(* IEC 61131-3 sources: lpmlv2022/test, 9 files *)

(* ---- test.st ---- *)
USING AxUnit.Assert;

NAMESPACE Simatic.Ax.lpmlv2022.Tests
    {TestFixture}
    CLASS MyTestFixture
        {Test}
        METHOD PUBLIC MyTestMethod
            Equal(actual := TRUE, expected := TRUE);
        END_METHOD
    END_CLASS
END_NAMESPACE

(* ---- TestConfigureCompleteCmdCfg.st ---- *)
USING AxUnit;
USING Simatic.Ax.LPMLV2022;

NAMESPACE Simatic.Ax.LPMLV2022.Tests

    {TestFixture}
    CLASS TestConfigureCompleteCmdCfg

        {Test}
        METHOD PUBLIC TestOnlySuspended
            VAR_TEMP
                result : DWORD;
            END_VAR

            ConfigureCompleteCmdCfg(
                Suspended := TRUE,
                Execute := FALSE,
                Held := FALSE,
                completeCmdCfg => result);

            Assert.Equal(actual := result.%X5, expected := TRUE);
            Assert.Equal(actual := result.%X6, expected := FALSE);
            Assert.Equal(actual := result.%X11, expected := FALSE);
            // Verify expected DWORD value (bit 5 set = 2^5 = 32 = 16#20)
            Assert.Equal(actual := result, expected := DWORD#16#0000_0020);

        END_METHOD

        {Test}
        METHOD PUBLIC TestOnlyExecute
            VAR_TEMP
                result : DWORD;
            END_VAR

            ConfigureCompleteCmdCfg(
                Suspended := FALSE,
                Execute := TRUE,
                Held := FALSE,
                completeCmdCfg => result);

            Assert.Equal(actual := result.%X5, expected := FALSE);
            Assert.Equal(actual := result.%X6, expected := TRUE);
            Assert.Equal(actual := result.%X11, expected := FALSE);
            // Verify expected DWORD value (bit 6 set = 2^6 = 64 = 16#40)
            Assert.Equal(actual := result, expected := DWORD#16#0000_0040);

        END_METHOD

        {Test}
        METHOD PUBLIC TestOnlyHeld
            VAR_TEMP
                result : DWORD;
            END_VAR

            ConfigureCompleteCmdCfg(
                Suspended := FALSE,
                Execute := FALSE,
                Held := TRUE,
                completeCmdCfg => result);

            Assert.Equal(actual := result.%X5, expected := FALSE);
            Assert.Equal(actual := result.%X6, expected := FALSE);
            Assert.Equal(actual := result.%X11, expected := TRUE);
            // Verify expected DWORD value (bit 11 set = 2^11 = 2048 = 16#800)
            Assert.Equal(actual := result, expected := DWORD#16#0000_0800);

        END_METHOD

        {Test}
        METHOD PUBLIC TestSuspendedAndExecute
            VAR_TEMP
                result : DWORD;
            END_VAR

            ConfigureCompleteCmdCfg(
                Suspended := TRUE,
                Execute := TRUE,
                Held := FALSE,
                completeCmdCfg => result);

            Assert.Equal(actual := result.%X5, expected := TRUE);
            Assert.Equal(actual := result.%X6, expected := TRUE);
            Assert.Equal(actual := result.%X11, expected := FALSE);
            // Verify expected DWORD value (bits 5+6 set = 32+64 = 96 = 16#60)
            Assert.Equal(actual := result, expected := DWORD#16#0000_0060);

        END_METHOD

        {Test}
        METHOD PUBLIC TestSuspendedAndHeld
            VAR_TEMP
                result : DWORD;
            END_VAR

            ConfigureCompleteCmdCfg(
                Suspended := TRUE,
                Execute := FALSE,
                Held := TRUE,
                completeCmdCfg => result);

            Assert.Equal(actual := result.%X5, expected := TRUE);
            Assert.Equal(actual := result.%X6, expected := FALSE);
            Assert.Equal(actual := result.%X11, expected := TRUE);
            // Verify expected DWORD value (bits 5+11 set = 32+2048 = 2080 = 16#820)
            Assert.Equal(actual := result, expected := DWORD#16#0000_0820);

        END_METHOD

        {Test}
        METHOD PUBLIC TestExecuteAndHeld
            VAR_TEMP
                result : DWORD;
            END_VAR

            ConfigureCompleteCmdCfg(
                Suspended := FALSE,
                Execute := TRUE,
                Held := TRUE,
                completeCmdCfg => result);

            Assert.Equal(actual := result.%X5, expected := FALSE);
            Assert.Equal(actual := result.%X6, expected := TRUE);
            Assert.Equal(actual := result.%X11, expected := TRUE);
            // Verify expected DWORD value (bits 6+11 set = 64+2048 = 2112 = 16#840)
            Assert.Equal(actual := result, expected := DWORD#16#0000_0840);

        END_METHOD

        {Test}
        METHOD PUBLIC TestAllStatesEnabled
            VAR_TEMP
                result : DWORD;
            END_VAR

            ConfigureCompleteCmdCfg(
                Suspended := TRUE,
                Execute := TRUE,
                Held := TRUE,
                completeCmdCfg => result);

            Assert.Equal(actual := result.%X5, expected := TRUE);
            Assert.Equal(actual := result.%X6, expected := TRUE);
            Assert.Equal(actual := result.%X11, expected := TRUE);
            // Verify expected DWORD value (bits 5+6+11 set = 32+64+2048 = 2144 = 16#860)
            Assert.Equal(actual := result, expected := DWORD#16#0000_0860);

        END_METHOD

        {Test}
        METHOD PUBLIC TestAllStatesDisabled
            VAR_TEMP
                result : DWORD;
            END_VAR

            ConfigureCompleteCmdCfg(
                Suspended := FALSE,
                Execute := FALSE,
                Held := FALSE,
                completeCmdCfg => result);

            Assert.Equal(actual := result.%X5, expected := FALSE);
            Assert.Equal(actual := result.%X6, expected := FALSE);
            Assert.Equal(actual := result.%X11, expected := FALSE);
            // Verify expected DWORD value (no bits set = 0)
            Assert.Equal(actual := result, expected := DWORD#16#0000_0000);

        END_METHOD

        {Test}
        METHOD PUBLIC TestUnusedBitsRemainZero
            VAR_TEMP
                result : DWORD;
                i : INT;
            END_VAR

            ConfigureCompleteCmdCfg(
                Suspended := TRUE,
                Execute := TRUE,
                Held := TRUE,
                completeCmdCfg => result);

            // Test that only the expected bits (5, 6, 11) are set
            // and all other bits remain 0
            FOR i := 0 TO 31 DO
                IF i = 5 OR i = 6 OR i = 11 THEN
                    // These bits should be TRUE
                    CONTINUE;
                ELSE
                    // All other bits should be FALSE
                    CASE i OF
                        0: Assert.Equal(actual := result.%X0, expected := FALSE);
                        1: Assert.Equal(actual := result.%X1, expected := FALSE);
                        2: Assert.Equal(actual := result.%X2, expected := FALSE);
                        3: Assert.Equal(actual := result.%X3, expected := FALSE);
                        4: Assert.Equal(actual := result.%X4, expected := FALSE);
                        7: Assert.Equal(actual := result.%X7, expected := FALSE);
                        8: Assert.Equal(actual := result.%X8, expected := FALSE);
                        9: Assert.Equal(actual := result.%X9, expected := FALSE);
                        10: Assert.Equal(actual := result.%X10, expected := FALSE);
                        12: Assert.Equal(actual := result.%X12, expected := FALSE);
                        13: Assert.Equal(actual := result.%X13, expected := FALSE);
                        14: Assert.Equal(actual := result.%X14, expected := FALSE);
                        15: Assert.Equal(actual := result.%X15, expected := FALSE);
                        // Testing a few more significant bits
                        16: Assert.Equal(actual := result.%X16, expected := FALSE);
                        20: Assert.Equal(actual := result.%X20, expected := FALSE);
                        31: Assert.Equal(actual := result.%X31, expected := FALSE);
                    END_CASE;
                END_IF;
            END_FOR;

        END_METHOD
    END_CLASS

END_NAMESPACE

(* ---- TestConfigureDisabledStatesCfg.st ---- *)
USING AxUnit;
USING Simatic.Ax.LPMLV2022;

NAMESPACE Simatic.Ax.LPMLV2022.Tests

    {TestFixture}
    CLASS TestConfigureDisabledStatesCfg

        {Test}
        METHOD PUBLIC TestOnlyClearing
            VAR_TEMP
                result : DWORD;
            END_VAR

            ConfigureDisabledStatesCfg(
                Clearing := TRUE,
                Starting := FALSE,
                Suspended := FALSE,
                Stopping := FALSE,
                Aborting := FALSE,
                Holding := FALSE,
                Held := FALSE,
                Unholding := FALSE,
                Suspending := FALSE,
                Unsuspending := FALSE,
                Resetting := FALSE,
                Completing := FALSE,
                Completed := FALSE,
                DisabledStatesCfg => result);

            Assert.Equal(actual := result.%X1, expected := TRUE);
            Assert.Equal(actual := result.%X3, expected := FALSE);
            Assert.Equal(actual := result.%X5, expected := FALSE);
            // Verify expected DWORD value (bit 1 set = 2^1 = 2 = 16#02)
            Assert.Equal(actual := result, expected := DWORD#16#0000_0002);

        END_METHOD

        {Test}
        METHOD PUBLIC TestOnlyStarting
            VAR_TEMP
                result : DWORD;
            END_VAR

            ConfigureDisabledStatesCfg(
                Clearing := FALSE,
                Starting := TRUE,
                Suspended := FALSE,
                Stopping := FALSE,
                Aborting := FALSE,
                Holding := FALSE,
                Held := FALSE,
                Unholding := FALSE,
                Suspending := FALSE,
                Unsuspending := FALSE,
                Resetting := FALSE,
                Completing := FALSE,
                Completed := FALSE,
                DisabledStatesCfg => result);

            Assert.Equal(actual := result.%X1, expected := FALSE);
            Assert.Equal(actual := result.%X3, expected := TRUE);
            Assert.Equal(actual := result.%X5, expected := FALSE);
            // Verify expected DWORD value (bit 3 set = 2^3 = 8 = 16#08)
            Assert.Equal(actual := result, expected := DWORD#16#0000_0008);

        END_METHOD

        {Test}
        METHOD PUBLIC TestOnlySuspended
            VAR_TEMP
                result : DWORD;
            END_VAR

            ConfigureDisabledStatesCfg(
                Clearing := FALSE,
                Starting := FALSE,
                Suspended := TRUE,
                Stopping := FALSE,
                Aborting := FALSE,
                Holding := FALSE,
                Held := FALSE,
                Unholding := FALSE,
                Suspending := FALSE,
                Unsuspending := FALSE,
                Resetting := FALSE,
                Completing := FALSE,
                Completed := FALSE,
                DisabledStatesCfg => result);

            Assert.Equal(actual := result.%X5, expected := TRUE);
            // Verify expected DWORD value (bit 5 set = 2^5 = 32 = 16#20)
            Assert.Equal(actual := result, expected := DWORD#16#0000_0020);

        END_METHOD

        {Test}
        METHOD PUBLIC TestOnlyStopping
            VAR_TEMP
                result : DWORD;
            END_VAR

            ConfigureDisabledStatesCfg(
                Clearing := FALSE,
                Starting := FALSE,
                Suspended := FALSE,
                Stopping := TRUE,
                Aborting := FALSE,
                Holding := FALSE,
                Held := FALSE,
                Unholding := FALSE,
                Suspending := FALSE,
                Unsuspending := FALSE,
                Resetting := FALSE,
                Completing := FALSE,
                Completed := FALSE,
                DisabledStatesCfg => result);

            Assert.Equal(actual := result.%X7, expected := TRUE);
            // Verify expected DWORD value (bit 7 set = 2^7 = 128 = 16#80)
            Assert.Equal(actual := result, expected := DWORD#16#0000_0080);

        END_METHOD

        {Test}
        METHOD PUBLIC TestOnlyAborting
            VAR_TEMP
                result : DWORD;
            END_VAR

            ConfigureDisabledStatesCfg(
                Clearing := FALSE,
                Starting := FALSE,
                Suspended := FALSE,
                Stopping := FALSE,
                Aborting := TRUE,
                Holding := FALSE,
                Held := FALSE,
                Unholding := FALSE,
                Suspending := FALSE,
                Unsuspending := FALSE,
                Resetting := FALSE,
                Completing := FALSE,
                Completed := FALSE,
                DisabledStatesCfg => result);

            Assert.Equal(actual := result.%X8, expected := TRUE);
            // Verify expected DWORD value (bit 8 set = 2^8 = 256 = 16#100)
            Assert.Equal(actual := result, expected := DWORD#16#0000_0100);

        END_METHOD

        {Test}
        METHOD PUBLIC TestOnlyHolding
            VAR_TEMP
                result : DWORD;
            END_VAR

            ConfigureDisabledStatesCfg(
                Clearing := FALSE,
                Starting := FALSE,
                Suspended := FALSE,
                Stopping := FALSE,
                Aborting := FALSE,
                Holding := TRUE,
                Held := FALSE,
                Unholding := FALSE,
                Suspending := FALSE,
                Unsuspending := FALSE,
                Resetting := FALSE,
                Completing := FALSE,
                Completed := FALSE,
                DisabledStatesCfg => result);

            Assert.Equal(actual := result.%X10, expected := TRUE);
            // Verify expected DWORD value (bit 10 set = 2^10 = 1024 = 16#400)
            Assert.Equal(actual := result, expected := DWORD#16#0000_0400);

        END_METHOD

        {Test}
        METHOD PUBLIC TestOnlyHeld
            VAR_TEMP
                result : DWORD;
            END_VAR

            ConfigureDisabledStatesCfg(
                Clearing := FALSE,
                Starting := FALSE,
                Suspended := FALSE,
                Stopping := FALSE,
                Aborting := FALSE,
                Holding := FALSE,
                Held := TRUE,
                Unholding := FALSE,
                Suspending := FALSE,
                Unsuspending := FALSE,
                Resetting := FALSE,
                Completing := FALSE,
                Completed := FALSE,
                DisabledStatesCfg => result);

            Assert.Equal(actual := result.%X11, expected := TRUE);
            // Verify expected DWORD value (bit 11 set = 2^11 = 2048 = 16#800)
            Assert.Equal(actual := result, expected := DWORD#16#0000_0800);

        END_METHOD

        {Test}
        METHOD PUBLIC TestOnlyUnholding
            VAR_TEMP
                result : DWORD;
            END_VAR

            ConfigureDisabledStatesCfg(
                Clearing := FALSE,
                Starting := FALSE,
                Suspended := FALSE,
                Stopping := FALSE,
                Aborting := FALSE,
                Holding := FALSE,
                Held := FALSE,
                Unholding := TRUE,
                Suspending := FALSE,
                Unsuspending := FALSE,
                Resetting := FALSE,
                Completing := FALSE,
                Completed := FALSE,
                DisabledStatesCfg => result);

            Assert.Equal(actual := result.%X12, expected := TRUE);
            // Verify expected DWORD value (bit 12 set = 2^12 = 4096 = 16#1000)
            Assert.Equal(actual := result, expected := DWORD#16#0000_1000);

        END_METHOD

        {Test}
        METHOD PUBLIC TestOnlySuspending
            VAR_TEMP
                result : DWORD;
            END_VAR

            ConfigureDisabledStatesCfg(
                Clearing := FALSE,
                Starting := FALSE,
                Suspended := FALSE,
                Stopping := FALSE,
                Aborting := FALSE,
                Holding := FALSE,
                Held := FALSE,
                Unholding := FALSE,
                Suspending := TRUE,
                Unsuspending := FALSE,
                Resetting := FALSE,
                Completing := FALSE,
                Completed := FALSE,
                DisabledStatesCfg => result);

            Assert.Equal(actual := result.%X13, expected := TRUE);
            // Verify expected DWORD value (bit 13 set = 2^13 = 8192 = 16#2000)
            Assert.Equal(actual := result, expected := DWORD#16#0000_2000);

        END_METHOD

        {Test}
        METHOD PUBLIC TestOnlyUnsuspending
            VAR_TEMP
                result : DWORD;
            END_VAR

            ConfigureDisabledStatesCfg(
                Clearing := FALSE,
                Starting := FALSE,
                Suspended := FALSE,
                Stopping := FALSE,
                Aborting := FALSE,
                Holding := FALSE,
                Held := FALSE,
                Unholding := FALSE,
                Suspending := FALSE,
                Unsuspending := TRUE,
                Resetting := FALSE,
                Completing := FALSE,
                Completed := FALSE,
                DisabledStatesCfg => result);

            Assert.Equal(actual := result.%X14, expected := TRUE);
            // Verify expected DWORD value (bit 14 set = 2^14 = 16384 = 16#4000)
            Assert.Equal(actual := result, expected := DWORD#16#0000_4000);

        END_METHOD

        {Test}
        METHOD PUBLIC TestOnlyResetting
            VAR_TEMP
                result : DWORD;
            END_VAR

            ConfigureDisabledStatesCfg(
                Clearing := FALSE,
                Starting := FALSE,
                Suspended := FALSE,
                Stopping := FALSE,
                Aborting := FALSE,
                Holding := FALSE,
                Held := FALSE,
                Unholding := FALSE,
                Suspending := FALSE,
                Unsuspending := FALSE,
                Resetting := TRUE,
                Completing := FALSE,
                Completed := FALSE,
                DisabledStatesCfg => result);

            Assert.Equal(actual := result.%X15, expected := TRUE);
            // Verify expected DWORD value (bit 15 set = 2^15 = 32768 = 16#8000)
            Assert.Equal(actual := result, expected := DWORD#16#0000_8000);

        END_METHOD

        {Test}
        METHOD PUBLIC TestOnlyCompleting
            VAR_TEMP
                result : DWORD;
            END_VAR

            ConfigureDisabledStatesCfg(
                Clearing := FALSE,
                Starting := FALSE,
                Suspended := FALSE,
                Stopping := FALSE,
                Aborting := FALSE,
                Holding := FALSE,
                Held := FALSE,
                Unholding := FALSE,
                Suspending := FALSE,
                Unsuspending := FALSE,
                Resetting := FALSE,
                Completing := TRUE,
                Completed := FALSE,
                DisabledStatesCfg => result);

            Assert.Equal(actual := result.%X16, expected := TRUE);
            // Verify expected DWORD value (bit 16 set = 2^16 = 65536 = 16#10000)
            Assert.Equal(actual := result, expected := DWORD#16#0001_0000);

        END_METHOD

        {Test}
        METHOD PUBLIC TestOnlyCompleted
            VAR_TEMP
                result : DWORD;
            END_VAR

            ConfigureDisabledStatesCfg(
                Clearing := FALSE,
                Starting := FALSE,
                Suspended := FALSE,
                Stopping := FALSE,
                Aborting := FALSE,
                Holding := FALSE,
                Held := FALSE,
                Unholding := FALSE,
                Suspending := FALSE,
                Unsuspending := FALSE,
                Resetting := FALSE,
                Completing := FALSE,
                Completed := TRUE,
                DisabledStatesCfg => result);

            Assert.Equal(actual := result.%X17, expected := TRUE);
            // Verify expected DWORD value (bit 17 set = 2^17 = 131072 = 16#20000)
            Assert.Equal(actual := result, expected := DWORD#16#0002_0000);

        END_METHOD

        {Test}
        METHOD PUBLIC TestCombinationClearingAndStarting
            VAR_TEMP
                result : DWORD;
            END_VAR

            ConfigureDisabledStatesCfg(
                Clearing := TRUE,
                Starting := TRUE,
                Suspended := FALSE,
                Stopping := FALSE,
                Aborting := FALSE,
                Holding := FALSE,
                Held := FALSE,
                Unholding := FALSE,
                Suspending := FALSE,
                Unsuspending := FALSE,
                Resetting := FALSE,
                Completing := FALSE,
                Completed := FALSE,
                DisabledStatesCfg => result);

            Assert.Equal(actual := result.%X1, expected := TRUE);
            Assert.Equal(actual := result.%X3, expected := TRUE);
            // Verify expected DWORD value (bits 1+3 set = 2+8 = 10 = 16#0A)
            Assert.Equal(actual := result, expected := DWORD#16#0000_000A);

        END_METHOD

        {Test}
        METHOD PUBLIC TestCombinationHoldingStates
            VAR_TEMP
                result : DWORD;
            END_VAR

            ConfigureDisabledStatesCfg(
                Clearing := FALSE,
                Starting := FALSE,
                Suspended := FALSE,
                Stopping := FALSE,
                Aborting := FALSE,
                Holding := TRUE,
                Held := TRUE,
                Unholding := TRUE,
                Suspending := FALSE,
                Unsuspending := FALSE,
                Resetting := FALSE,
                Completing := FALSE,
                Completed := FALSE,
                DisabledStatesCfg => result);

            Assert.Equal(actual := result.%X10, expected := TRUE);
            Assert.Equal(actual := result.%X11, expected := TRUE);
            Assert.Equal(actual := result.%X12, expected := TRUE);
            // Verify expected DWORD value (bits 10+11+12 set = 1024+2048+4096 = 7168 = 16#1C00)
            Assert.Equal(actual := result, expected := DWORD#16#0000_1C00);

        END_METHOD

        {Test}
        METHOD PUBLIC TestAllStatesDisabled
            VAR_TEMP
                result : DWORD;
            END_VAR

            ConfigureDisabledStatesCfg(
                Clearing := TRUE,
                Starting := TRUE,
                Suspended := TRUE,
                Stopping := TRUE,
                Aborting := TRUE,
                Holding := TRUE,
                Held := TRUE,
                Unholding := TRUE,
                Suspending := TRUE,
                Unsuspending := TRUE,
                Resetting := TRUE,
                Completing := TRUE,
                Completed := TRUE,
                DisabledStatesCfg => result);

            // Verify all configured bits are set
            Assert.Equal(actual := result.%X1, expected := TRUE);   // Clearing
            Assert.Equal(actual := result.%X3, expected := TRUE);   // Starting
            Assert.Equal(actual := result.%X5, expected := TRUE);   // Suspended
            Assert.Equal(actual := result.%X7, expected := TRUE);   // Stopping
            Assert.Equal(actual := result.%X8, expected := TRUE);   // Aborting
            Assert.Equal(actual := result.%X10, expected := TRUE);  // Holding
            Assert.Equal(actual := result.%X11, expected := TRUE);  // Held
            Assert.Equal(actual := result.%X12, expected := TRUE);  // Unholding
            Assert.Equal(actual := result.%X13, expected := TRUE);  // Suspending
            Assert.Equal(actual := result.%X14, expected := TRUE);  // Unsuspending
            Assert.Equal(actual := result.%X15, expected := TRUE);  // Resetting
            Assert.Equal(actual := result.%X16, expected := TRUE);  // Completing
            Assert.Equal(actual := result.%X17, expected := TRUE);  // Completed

            // Verify expected DWORD value (all configured bits set)
            // bits 1,3,5,7,8,10,11,12,13,14,15,16,17 = 2+8+32+128+256+1024+2048+4096+8192+16384+32768+65536+131072 = 261546 = 16#3FDAA
            Assert.Equal(actual := result, expected := DWORD#16#0003_FDAA);

        END_METHOD

        {Test}
        METHOD PUBLIC TestAllStatesEnabled
            VAR_TEMP
                result : DWORD;
            END_VAR

            ConfigureDisabledStatesCfg(
                Clearing := FALSE,
                Starting := FALSE,
                Suspended := FALSE,
                Stopping := FALSE,
                Aborting := FALSE,
                Holding := FALSE,
                Held := FALSE,
                Unholding := FALSE,
                Suspending := FALSE,
                Unsuspending := FALSE,
                Resetting := FALSE,
                Completing := FALSE,
                Completed := FALSE,
                DisabledStatesCfg => result);

            // Verify all configured bits are FALSE (states enabled)
            Assert.Equal(actual := result.%X1, expected := FALSE);
            Assert.Equal(actual := result.%X3, expected := FALSE);
            Assert.Equal(actual := result.%X5, expected := FALSE);
            Assert.Equal(actual := result.%X7, expected := FALSE);
            Assert.Equal(actual := result.%X8, expected := FALSE);
            Assert.Equal(actual := result.%X10, expected := FALSE);
            Assert.Equal(actual := result.%X11, expected := FALSE);
            Assert.Equal(actual := result.%X12, expected := FALSE);
            Assert.Equal(actual := result.%X13, expected := FALSE);
            Assert.Equal(actual := result.%X14, expected := FALSE);
            Assert.Equal(actual := result.%X15, expected := FALSE);
            Assert.Equal(actual := result.%X16, expected := FALSE);
            Assert.Equal(actual := result.%X17, expected := FALSE);

            // Verify expected DWORD value (no bits set = 0)
            Assert.Equal(actual := result, expected := DWORD#16#0000_0000);

        END_METHOD

        {Test}
        METHOD PUBLIC TestAlwaysPresentBitsRemainUnaffected
            VAR_TEMP
                result : DWORD;
            END_VAR

            // Test with all states disabled to verify that always-present bits (2,4,6,9) remain 0
            ConfigureDisabledStatesCfg(
                Clearing := TRUE,
                Starting := TRUE,
                Suspended := TRUE,
                Stopping := TRUE,
                Aborting := TRUE,
                Holding := TRUE,
                Held := TRUE,
                Unholding := TRUE,
                Suspending := TRUE,
                Unsuspending := TRUE,
                Resetting := TRUE,
                Completing := TRUE,
                Completed := TRUE,
                DisabledStatesCfg => result);

            // Verify that the always-present states (Stopped, Idle, Execute, Aborted)
            // remain FALSE as they cannot be disabled according to the comment
            Assert.Equal(actual := result.%X2, expected := FALSE);  // Stopped - always present
            Assert.Equal(actual := result.%X4, expected := FALSE);  // Idle - always present
            Assert.Equal(actual := result.%X6, expected := FALSE);  // Execute - always present
            Assert.Equal(actual := result.%X9, expected := FALSE);  // Aborted - always present

        END_METHOD

        {Test}
        METHOD PUBLIC TestUnusedBitsRemainZero
            VAR_TEMP
                result : DWORD;
            END_VAR

            // Test with all configurable states disabled
            ConfigureDisabledStatesCfg(
                Clearing := TRUE,
                Starting := TRUE,
                Suspended := TRUE,
                Stopping := TRUE,
                Aborting := TRUE,
                Holding := TRUE,
                Held := TRUE,
                Unholding := TRUE,
                Suspending := TRUE,
                Unsuspending := TRUE,
                Resetting := TRUE,
                Completing := TRUE,
                Completed := TRUE,
                DisabledStatesCfg => result);

            // Test that unused bits remain 0
            Assert.Equal(actual := result.%X0, expected := FALSE);   // Unused
            Assert.Equal(actual := result.%X18, expected := FALSE);  // Unused
            Assert.Equal(actual := result.%X19, expected := FALSE);  // Unused
            Assert.Equal(actual := result.%X20, expected := FALSE);  // Unused
            Assert.Equal(actual := result.%X25, expected := FALSE);  // Unused
            Assert.Equal(actual := result.%X31, expected := FALSE);  // Unused (MSB)

        END_METHOD

    END_CLASS

END_NAMESPACE

(* ---- TestConfigureEnabledModesCfg.st ---- *)
USING AxUnit;
USING Simatic.Ax.LPMLV2022;

NAMESPACE Simatic.Ax.LPMLV2022.Tests

    {TestFixture}
    CLASS TestConfigureEnabledModesCfg

        {Test}
        METHOD PUBLIC TestOnlyMandatoryManualMode
            VAR_TEMP
                result : DWORD;
            END_VAR

            ConfigureEnabledModesCfg(
                ProductionMode := FALSE,
                MaintenanceMode := FALSE,
                UserMode01 := FALSE, UserMode02 := FALSE, UserMode03 := FALSE, UserMode04 := FALSE, UserMode05 := FALSE,
                UserMode06 := FALSE, UserMode07 := FALSE, UserMode08 := FALSE, UserMode09 := FALSE, UserMode10 := FALSE,
                UserMode11 := FALSE, UserMode12 := FALSE, UserMode13 := FALSE, UserMode14 := FALSE, UserMode15 := FALSE,
                UserMode16 := FALSE, UserMode17 := FALSE, UserMode18 := FALSE, UserMode19 := FALSE, UserMode20 := FALSE,
                UserMode21 := FALSE, UserMode22 := FALSE, UserMode23 := FALSE, UserMode24 := FALSE, UserMode25 := FALSE,
                UserMode26 := FALSE, UserMode27 := FALSE, UserMode28 := FALSE,
                EnabledModesCfg => result);

            // Verify only Manual mode (bit 3) is set
            Assert.Equal(actual := result.%X1, expected := FALSE);  // ProductionMode
            Assert.Equal(actual := result.%X2, expected := FALSE);  // MaintenanceMode
            Assert.Equal(actual := result.%X3, expected := TRUE);   // Manual mode (mandatory)
            Assert.Equal(actual := result.%X4, expected := FALSE);  // UserMode01

            // Verify expected DWORD value (only bit 3 set = 2^3 = 8 = 16#08)
            Assert.Equal(actual := result, expected := DWORD#16#0000_0008);

        END_METHOD

        {Test}
        METHOD PUBLIC TestOnlyProductionMode
            VAR_TEMP
                result : DWORD;
            END_VAR

            ConfigureEnabledModesCfg(
                ProductionMode := TRUE,
                MaintenanceMode := FALSE,
                UserMode01 := FALSE, UserMode02 := FALSE, UserMode03 := FALSE, UserMode04 := FALSE, UserMode05 := FALSE,
                UserMode06 := FALSE, UserMode07 := FALSE, UserMode08 := FALSE, UserMode09 := FALSE, UserMode10 := FALSE,
                UserMode11 := FALSE, UserMode12 := FALSE, UserMode13 := FALSE, UserMode14 := FALSE, UserMode15 := FALSE,
                UserMode16 := FALSE, UserMode17 := FALSE, UserMode18 := FALSE, UserMode19 := FALSE, UserMode20 := FALSE,
                UserMode21 := FALSE, UserMode22 := FALSE, UserMode23 := FALSE, UserMode24 := FALSE, UserMode25 := FALSE,
                UserMode26 := FALSE, UserMode27 := FALSE, UserMode28 := FALSE,
                EnabledModesCfg => result);

            Assert.Equal(actual := result.%X1, expected := TRUE);   // ProductionMode
            Assert.Equal(actual := result.%X2, expected := FALSE);  // MaintenanceMode
            Assert.Equal(actual := result.%X3, expected := TRUE);   // Manual mode (mandatory)

            // Verify expected DWORD value (bits 1+3 set = 2+8 = 10 = 16#0A)
            Assert.Equal(actual := result, expected := DWORD#16#0000_000A);

        END_METHOD

        {Test}
        METHOD PUBLIC TestOnlyMaintenanceMode
            VAR_TEMP
                result : DWORD;
            END_VAR

            ConfigureEnabledModesCfg(
                ProductionMode := FALSE,
                MaintenanceMode := TRUE,
                UserMode01 := FALSE, UserMode02 := FALSE, UserMode03 := FALSE, UserMode04 := FALSE, UserMode05 := FALSE,
                UserMode06 := FALSE, UserMode07 := FALSE, UserMode08 := FALSE, UserMode09 := FALSE, UserMode10 := FALSE,
                UserMode11 := FALSE, UserMode12 := FALSE, UserMode13 := FALSE, UserMode14 := FALSE, UserMode15 := FALSE,
                UserMode16 := FALSE, UserMode17 := FALSE, UserMode18 := FALSE, UserMode19 := FALSE, UserMode20 := FALSE,
                UserMode21 := FALSE, UserMode22 := FALSE, UserMode23 := FALSE, UserMode24 := FALSE, UserMode25 := FALSE,
                UserMode26 := FALSE, UserMode27 := FALSE, UserMode28 := FALSE,
                EnabledModesCfg => result);

            Assert.Equal(actual := result.%X1, expected := FALSE);  // ProductionMode
            Assert.Equal(actual := result.%X2, expected := TRUE);   // MaintenanceMode
            Assert.Equal(actual := result.%X3, expected := TRUE);   // Manual mode (mandatory)

            // Verify expected DWORD value (bits 2+3 set = 4+8 = 12 = 16#0C)
            Assert.Equal(actual := result, expected := DWORD#16#0000_000C);

        END_METHOD

        {Test}
        METHOD PUBLIC TestProductionAndMaintenanceModes
            VAR_TEMP
                result : DWORD;
            END_VAR

            ConfigureEnabledModesCfg(
                ProductionMode := TRUE,
                MaintenanceMode := TRUE,
                UserMode01 := FALSE, UserMode02 := FALSE, UserMode03 := FALSE, UserMode04 := FALSE, UserMode05 := FALSE,
                UserMode06 := FALSE, UserMode07 := FALSE, UserMode08 := FALSE, UserMode09 := FALSE, UserMode10 := FALSE,
                UserMode11 := FALSE, UserMode12 := FALSE, UserMode13 := FALSE, UserMode14 := FALSE, UserMode15 := FALSE,
                UserMode16 := FALSE, UserMode17 := FALSE, UserMode18 := FALSE, UserMode19 := FALSE, UserMode20 := FALSE,
                UserMode21 := FALSE, UserMode22 := FALSE, UserMode23 := FALSE, UserMode24 := FALSE, UserMode25 := FALSE,
                UserMode26 := FALSE, UserMode27 := FALSE, UserMode28 := FALSE,
                EnabledModesCfg => result);

            Assert.Equal(actual := result.%X1, expected := TRUE);   // ProductionMode
            Assert.Equal(actual := result.%X2, expected := TRUE);   // MaintenanceMode
            Assert.Equal(actual := result.%X3, expected := TRUE);   // Manual mode (mandatory)

            // Verify expected DWORD value (bits 1+2+3 set = 2+4+8 = 14 = 16#0E)
            Assert.Equal(actual := result, expected := DWORD#16#0000_000E);

        END_METHOD

        {Test}
        METHOD PUBLIC TestFirstFewUserModes
            VAR_TEMP
                result : DWORD;
            END_VAR

            ConfigureEnabledModesCfg(
                ProductionMode := FALSE,
                MaintenanceMode := FALSE,
                UserMode01 := TRUE, UserMode02 := TRUE, UserMode03 := TRUE, UserMode04 := FALSE, UserMode05 := FALSE,
                UserMode06 := FALSE, UserMode07 := FALSE, UserMode08 := FALSE, UserMode09 := FALSE, UserMode10 := FALSE,
                UserMode11 := FALSE, UserMode12 := FALSE, UserMode13 := FALSE, UserMode14 := FALSE, UserMode15 := FALSE,
                UserMode16 := FALSE, UserMode17 := FALSE, UserMode18 := FALSE, UserMode19 := FALSE, UserMode20 := FALSE,
                UserMode21 := FALSE, UserMode22 := FALSE, UserMode23 := FALSE, UserMode24 := FALSE, UserMode25 := FALSE,
                UserMode26 := FALSE, UserMode27 := FALSE, UserMode28 := FALSE,
                EnabledModesCfg => result);

            Assert.Equal(actual := result.%X3, expected := TRUE);   // Manual mode (mandatory)
            Assert.Equal(actual := result.%X4, expected := TRUE);   // UserMode01
            Assert.Equal(actual := result.%X5, expected := TRUE);   // UserMode02
            Assert.Equal(actual := result.%X6, expected := TRUE);   // UserMode03
            Assert.Equal(actual := result.%X7, expected := FALSE);  // UserMode04

            // Verify expected DWORD value (bits 3+4+5+6 set = 8+16+32+64 = 120 = 16#78)
            Assert.Equal(actual := result, expected := DWORD#16#0000_0078);

        END_METHOD

        {Test}
        METHOD PUBLIC TestLastFewUserModes
            VAR_TEMP
                result : DWORD;
            END_VAR

            ConfigureEnabledModesCfg(
                ProductionMode := FALSE,
                MaintenanceMode := FALSE,
                UserMode01 := FALSE, UserMode02 := FALSE, UserMode03 := FALSE, UserMode04 := FALSE, UserMode05 := FALSE,
                UserMode06 := FALSE, UserMode07 := FALSE, UserMode08 := FALSE, UserMode09 := FALSE, UserMode10 := FALSE,
                UserMode11 := FALSE, UserMode12 := FALSE, UserMode13 := FALSE, UserMode14 := FALSE, UserMode15 := FALSE,
                UserMode16 := FALSE, UserMode17 := FALSE, UserMode18 := FALSE, UserMode19 := FALSE, UserMode20 := FALSE,
                UserMode21 := FALSE, UserMode22 := FALSE, UserMode23 := FALSE, UserMode24 := FALSE, UserMode25 := FALSE,
                UserMode26 := TRUE, UserMode27 := TRUE, UserMode28 := TRUE,
                EnabledModesCfg => result);

            Assert.Equal(actual := result.%X3, expected := TRUE);   // Manual mode (mandatory)
            Assert.Equal(actual := result.%X29, expected := TRUE);  // UserMode26
            Assert.Equal(actual := result.%X30, expected := TRUE);  // UserMode27
            Assert.Equal(actual := result.%X31, expected := TRUE);  // UserMode28

            // Verify expected DWORD value (bits 3+29+30+31 set = 8+536870912+1073741824+2147483648 = 3757465592 = 16#E0000008)
            Assert.Equal(actual := result, expected := DWORD#16#E000_0008);

        END_METHOD

        {Test}
        METHOD PUBLIC TestMiddleUserModes
            VAR_TEMP
                result : DWORD;
            END_VAR

            ConfigureEnabledModesCfg(
                ProductionMode := FALSE,
                MaintenanceMode := FALSE,
                UserMode01 := FALSE, UserMode02 := FALSE, UserMode03 := FALSE, UserMode04 := FALSE, UserMode05 := FALSE,
                UserMode06 := FALSE, UserMode07 := FALSE, UserMode08 := FALSE, UserMode09 := FALSE, UserMode10 := FALSE,
                UserMode11 := FALSE, UserMode12 := FALSE, UserMode13 := TRUE, UserMode14 := TRUE, UserMode15 := TRUE,
                UserMode16 := FALSE, UserMode17 := FALSE, UserMode18 := FALSE, UserMode19 := FALSE, UserMode20 := FALSE,
                UserMode21 := FALSE, UserMode22 := FALSE, UserMode23 := FALSE, UserMode24 := FALSE, UserMode25 := FALSE,
                UserMode26 := FALSE, UserMode27 := FALSE, UserMode28 := FALSE,
                EnabledModesCfg => result);

            Assert.Equal(actual := result.%X3, expected := TRUE);   // Manual mode (mandatory)
            Assert.Equal(actual := result.%X16, expected := TRUE);  // UserMode13
            Assert.Equal(actual := result.%X17, expected := TRUE);  // UserMode14
            Assert.Equal(actual := result.%X18, expected := TRUE);  // UserMode15

            // Verify expected DWORD value (bits 3+16+17+18 set = 8+65536+131072+262144 = 458760 = 16#70008)
            Assert.Equal(actual := result, expected := DWORD#16#0007_0008);

        END_METHOD

        {Test}
        METHOD PUBLIC TestEveryOtherUserMode
            VAR_TEMP
                result : DWORD;
            END_VAR

            ConfigureEnabledModesCfg(
                ProductionMode := FALSE,
                MaintenanceMode := FALSE,
                UserMode01 := TRUE, UserMode02 := FALSE, UserMode03 := TRUE, UserMode04 := FALSE, UserMode05 := TRUE,
                UserMode06 := FALSE, UserMode07 := TRUE, UserMode08 := FALSE, UserMode09 := TRUE, UserMode10 := FALSE,
                UserMode11 := TRUE, UserMode12 := FALSE, UserMode13 := TRUE, UserMode14 := FALSE, UserMode15 := TRUE,
                UserMode16 := FALSE, UserMode17 := TRUE, UserMode18 := FALSE, UserMode19 := TRUE, UserMode20 := FALSE,
                UserMode21 := TRUE, UserMode22 := FALSE, UserMode23 := TRUE, UserMode24 := FALSE, UserMode25 := TRUE,
                UserMode26 := FALSE, UserMode27 := TRUE, UserMode28 := FALSE,
                EnabledModesCfg => result);

            Assert.Equal(actual := result.%X3, expected := TRUE);   // Manual mode (mandatory)
            Assert.Equal(actual := result.%X4, expected := TRUE);   // UserMode01
            Assert.Equal(actual := result.%X5, expected := FALSE);  // UserMode02
            Assert.Equal(actual := result.%X6, expected := TRUE);   // UserMode03
            Assert.Equal(actual := result.%X7, expected := FALSE);  // UserMode04
            Assert.Equal(actual := result.%X30, expected := TRUE);  // UserMode27
            Assert.Equal(actual := result.%X31, expected := FALSE); // UserMode28

            // Verify expected DWORD value (alternating pattern + mandatory bit 3)
            Assert.Equal(actual := result, expected := DWORD#16#5555_5558);

        END_METHOD

        {Test}
        METHOD PUBLIC TestAllModesEnabled
            VAR_TEMP
                result : DWORD;
            END_VAR

            ConfigureEnabledModesCfg(
                ProductionMode := TRUE,
                MaintenanceMode := TRUE,
                UserMode01 := TRUE, UserMode02 := TRUE, UserMode03 := TRUE, UserMode04 := TRUE, UserMode05 := TRUE,
                UserMode06 := TRUE, UserMode07 := TRUE, UserMode08 := TRUE, UserMode09 := TRUE, UserMode10 := TRUE,
                UserMode11 := TRUE, UserMode12 := TRUE, UserMode13 := TRUE, UserMode14 := TRUE, UserMode15 := TRUE,
                UserMode16 := TRUE, UserMode17 := TRUE, UserMode18 := TRUE, UserMode19 := TRUE, UserMode20 := TRUE,
                UserMode21 := TRUE, UserMode22 := TRUE, UserMode23 := TRUE, UserMode24 := TRUE, UserMode25 := TRUE,
                UserMode26 := TRUE, UserMode27 := TRUE, UserMode28 := TRUE,
                EnabledModesCfg => result);

            // Verify all configurable bits are set
            Assert.Equal(actual := result.%X1, expected := TRUE);   // ProductionMode
            Assert.Equal(actual := result.%X2, expected := TRUE);   // MaintenanceMode
            Assert.Equal(actual := result.%X3, expected := TRUE);   // Manual mode (mandatory)
            Assert.Equal(actual := result.%X4, expected := TRUE);   // UserMode01
            Assert.Equal(actual := result.%X31, expected := TRUE);  // UserMode28

            // Verify expected DWORD value (all bits 1-31 set except bit 0 = 0xFFFFFFFE)
            Assert.Equal(actual := result, expected := DWORD#16#FFFF_FFFE);

        END_METHOD

        {Test}
        METHOD PUBLIC TestMandatoryBitAlwaysSet
            VAR_TEMP
                result : DWORD;
            END_VAR

            // Test different combinations to ensure Manual mode (bit 3) is always set

            // Test 1: All modes disabled
            ConfigureEnabledModesCfg(
                ProductionMode := FALSE,
                MaintenanceMode := FALSE,
                UserMode01 := FALSE, UserMode02 := FALSE, UserMode03 := FALSE, UserMode04 := FALSE, UserMode05 := FALSE,
                UserMode06 := FALSE, UserMode07 := FALSE, UserMode08 := FALSE, UserMode09 := FALSE, UserMode10 := FALSE,
                UserMode11 := FALSE, UserMode12 := FALSE, UserMode13 := FALSE, UserMode14 := FALSE, UserMode15 := FALSE,
                UserMode16 := FALSE, UserMode17 := FALSE, UserMode18 := FALSE, UserMode19 := FALSE, UserMode20 := FALSE,
                UserMode21 := FALSE, UserMode22 := FALSE, UserMode23 := FALSE, UserMode24 := FALSE, UserMode25 := FALSE,
                UserMode26 := FALSE, UserMode27 := FALSE, UserMode28 := FALSE,
                EnabledModesCfg => result);

            Assert.Equal(actual := result.%X3, expected := TRUE);   // Manual mode must be set

            // Test 2: Only Production enabled
            ConfigureEnabledModesCfg(
                ProductionMode := TRUE,
                MaintenanceMode := FALSE,
                UserMode01 := FALSE, UserMode02 := FALSE, UserMode03 := FALSE, UserMode04 := FALSE, UserMode05 := FALSE,
                UserMode06 := FALSE, UserMode07 := FALSE, UserMode08 := FALSE, UserMode09 := FALSE, UserMode10 := FALSE,
                UserMode11 := FALSE, UserMode12 := FALSE, UserMode13 := FALSE, UserMode14 := FALSE, UserMode15 := FALSE,
                UserMode16 := FALSE, UserMode17 := FALSE, UserMode18 := FALSE, UserMode19 := FALSE, UserMode20 := FALSE,
                UserMode21 := FALSE, UserMode22 := FALSE, UserMode23 := FALSE, UserMode24 := FALSE, UserMode25 := FALSE,
                UserMode26 := FALSE, UserMode27 := FALSE, UserMode28 := FALSE,
                EnabledModesCfg => result);

            Assert.Equal(actual := result.%X3, expected := TRUE);   // Manual mode must be set

        END_METHOD

        {Test}
        METHOD PUBLIC TestUnusedBitZero
            VAR_TEMP
                result : DWORD;
            END_VAR

            // Test with all modes enabled to verify bit 0 remains unused
            ConfigureEnabledModesCfg(
                ProductionMode := TRUE,
                MaintenanceMode := TRUE,
                UserMode01 := TRUE, UserMode02 := TRUE, UserMode03 := TRUE, UserMode04 := TRUE, UserMode05 := TRUE,
                UserMode06 := TRUE, UserMode07 := TRUE, UserMode08 := TRUE, UserMode09 := TRUE, UserMode10 := TRUE,
                UserMode11 := TRUE, UserMode12 := TRUE, UserMode13 := TRUE, UserMode14 := TRUE, UserMode15 := TRUE,
                UserMode16 := TRUE, UserMode17 := TRUE, UserMode18 := TRUE, UserMode19 := TRUE, UserMode20 := TRUE,
                UserMode21 := TRUE, UserMode22 := TRUE, UserMode23 := TRUE, UserMode24 := TRUE, UserMode25 := TRUE,
                UserMode26 := TRUE, UserMode27 := TRUE, UserMode28 := TRUE,
                EnabledModesCfg => result);

            // Verify bit 0 is not used and remains FALSE
            Assert.Equal(actual := result.%X0, expected := FALSE);

        END_METHOD

        {Test}
        METHOD PUBLIC TestBitMappingVerification
            VAR_TEMP
                result : DWORD;
            END_VAR

            // Test specific bit mappings by enabling only one mode at a time

            // Test UserMode01 -> bit 4
            ConfigureEnabledModesCfg(
                ProductionMode := FALSE,
                MaintenanceMode := FALSE,
                UserMode01 := TRUE, UserMode02 := FALSE, UserMode03 := FALSE, UserMode04 := FALSE, UserMode05 := FALSE,
                UserMode06 := FALSE, UserMode07 := FALSE, UserMode08 := FALSE, UserMode09 := FALSE, UserMode10 := FALSE,
                UserMode11 := FALSE, UserMode12 := FALSE, UserMode13 := FALSE, UserMode14 := FALSE, UserMode15 := FALSE,
                UserMode16 := FALSE, UserMode17 := FALSE, UserMode18 := FALSE, UserMode19 := FALSE, UserMode20 := FALSE,
                UserMode21 := FALSE, UserMode22 := FALSE, UserMode23 := FALSE, UserMode24 := FALSE, UserMode25 := FALSE,
                UserMode26 := FALSE, UserMode27 := FALSE, UserMode28 := FALSE,
                EnabledModesCfg => result);

            Assert.Equal(actual := result.%X4, expected := TRUE);   // UserMode01 -> bit 4
            Assert.Equal(actual := result.%X5, expected := FALSE);  // UserMode02 -> bit 5 (should be false)

            // Verify expected DWORD value (bits 3+4 set = 8+16 = 24 = 16#18)
            Assert.Equal(actual := result, expected := DWORD#16#0000_0018);

        END_METHOD

        {Test}
        METHOD PUBLIC TestHighOrderBitMapping
            VAR_TEMP
                result : DWORD;
            END_VAR

            // Test high-order bit mappings
            ConfigureEnabledModesCfg(
                ProductionMode := FALSE,
                MaintenanceMode := FALSE,
                UserMode01 := FALSE, UserMode02 := FALSE, UserMode03 := FALSE, UserMode04 := FALSE, UserMode05 := FALSE,
                UserMode06 := FALSE, UserMode07 := FALSE, UserMode08 := FALSE, UserMode09 := FALSE, UserMode10 := FALSE,
                UserMode11 := FALSE, UserMode12 := FALSE, UserMode13 := FALSE, UserMode14 := FALSE, UserMode15 := FALSE,
                UserMode16 := FALSE, UserMode17 := FALSE, UserMode18 := FALSE, UserMode19 := FALSE, UserMode20 := FALSE,
                UserMode21 := FALSE, UserMode22 := FALSE, UserMode23 := FALSE, UserMode24 := FALSE, UserMode25 := FALSE,
                UserMode26 := FALSE, UserMode27 := FALSE, UserMode28 := TRUE,
                EnabledModesCfg => result);

            Assert.Equal(actual := result.%X31, expected := TRUE);  // UserMode28 -> bit 31 (MSB)
            Assert.Equal(actual := result.%X30, expected := FALSE); // UserMode27 -> bit 30 (should be false)

            // Verify expected DWORD value (bits 3+31 set = 8+2147483648 = 2147483656 = 16#80000008)
            Assert.Equal(actual := result, expected := DWORD#16#8000_0008);

        END_METHOD

        {Test}
        METHOD PUBLIC TestSequentialUserModes
            VAR_TEMP
                result : DWORD;
            END_VAR

            // Test first 5 user modes to verify sequential bit mapping
            ConfigureEnabledModesCfg(
                ProductionMode := FALSE,
                MaintenanceMode := FALSE,
                UserMode01 := TRUE, UserMode02 := TRUE, UserMode03 := TRUE, UserMode04 := TRUE, UserMode05 := TRUE,
                UserMode06 := FALSE, UserMode07 := FALSE, UserMode08 := FALSE, UserMode09 := FALSE, UserMode10 := FALSE,
                UserMode11 := FALSE, UserMode12 := FALSE, UserMode13 := FALSE, UserMode14 := FALSE, UserMode15 := FALSE,
                UserMode16 := FALSE, UserMode17 := FALSE, UserMode18 := FALSE, UserMode19 := FALSE, UserMode20 := FALSE,
                UserMode21 := FALSE, UserMode22 := FALSE, UserMode23 := FALSE, UserMode24 := FALSE, UserMode25 := FALSE,
                UserMode26 := FALSE, UserMode27 := FALSE, UserMode28 := FALSE,
                EnabledModesCfg => result);

            Assert.Equal(actual := result.%X4, expected := TRUE);   // UserMode01 -> bit 4
            Assert.Equal(actual := result.%X5, expected := TRUE);   // UserMode02 -> bit 5
            Assert.Equal(actual := result.%X6, expected := TRUE);   // UserMode03 -> bit 6
            Assert.Equal(actual := result.%X7, expected := TRUE);   // UserMode04 -> bit 7
            Assert.Equal(actual := result.%X8, expected := TRUE);   // UserMode05 -> bit 8
            Assert.Equal(actual := result.%X9, expected := FALSE);  // UserMode06 -> bit 9 (should be false)

            // Verify expected DWORD value (bits 3+4+5+6+7+8 set = 8+16+32+64+128+256 = 504 = 16#1F8)
            Assert.Equal(actual := result, expected := DWORD#16#0000_01F8);

        END_METHOD

    END_CLASS

END_NAMESPACE

(* ---- TestConfigureHoldCmdCfg.st ---- *)
USING AxUnit;
USING Simatic.Ax.LPMLV2022;

NAMESPACE Simatic.Ax.LPMLV2022.Tests

    {TestFixture}
    CLASS TestConfigureHoldCmdCfg

        {Test}
        METHOD PUBLIC TestOnlyStarting
            VAR_TEMP
                result : DWORD;
            END_VAR

            ConfigureHoldCmdCfg(
                Starting := TRUE,
                Idle := FALSE,
                Suspended := FALSE,
                Execute := FALSE,
                Unholding := FALSE,
                Suspending := FALSE,
                Unsuspending := FALSE,
                Completing := FALSE,
                Completed := FALSE,
                holdCmdCfg => result);

            Assert.Equal(actual := result.%X3, expected := TRUE);
            Assert.Equal(actual := result.%X4, expected := FALSE);
            Assert.Equal(actual := result.%X5, expected := FALSE);
            Assert.Equal(actual := result.%X6, expected := FALSE);
            // Verify expected DWORD value (bit 3 set = 2^3 = 8 = 16#08)
            Assert.Equal(actual := result, expected := DWORD#16#0000_0008);

        END_METHOD

        {Test}
        METHOD PUBLIC TestOnlyIdle
            VAR_TEMP
                result : DWORD;
            END_VAR

            ConfigureHoldCmdCfg(
                Starting := FALSE,
                Idle := TRUE,
                Suspended := FALSE,
                Execute := FALSE,
                Unholding := FALSE,
                Suspending := FALSE,
                Unsuspending := FALSE,
                Completing := FALSE,
                Completed := FALSE,
                holdCmdCfg => result);

            Assert.Equal(actual := result.%X3, expected := FALSE);
            Assert.Equal(actual := result.%X4, expected := TRUE);
            Assert.Equal(actual := result.%X5, expected := FALSE);
            // Verify expected DWORD value (bit 4 set = 2^4 = 16 = 16#10)
            Assert.Equal(actual := result, expected := DWORD#16#0000_0010);

        END_METHOD

        {Test}
        METHOD PUBLIC TestOnlySuspended
            VAR_TEMP
                result : DWORD;
            END_VAR

            ConfigureHoldCmdCfg(
                Starting := FALSE,
                Idle := FALSE,
                Suspended := TRUE,
                Execute := FALSE,
                Unholding := FALSE,
                Suspending := FALSE,
                Unsuspending := FALSE,
                Completing := FALSE,
                Completed := FALSE,
                holdCmdCfg => result);

            Assert.Equal(actual := result.%X5, expected := TRUE);
            Assert.Equal(actual := result.%X6, expected := FALSE);
            // Verify expected DWORD value (bit 5 set = 2^5 = 32 = 16#20)
            Assert.Equal(actual := result, expected := DWORD#16#0000_0020);

        END_METHOD

        {Test}
        METHOD PUBLIC TestOnlyExecute
            VAR_TEMP
                result : DWORD;
            END_VAR

            ConfigureHoldCmdCfg(
                Starting := FALSE,
                Idle := FALSE,
                Suspended := FALSE,
                Execute := TRUE,
                Unholding := FALSE,
                Suspending := FALSE,
                Unsuspending := FALSE,
                Completing := FALSE,
                Completed := FALSE,
                holdCmdCfg => result);

            Assert.Equal(actual := result.%X6, expected := TRUE);
            Assert.Equal(actual := result.%X5, expected := FALSE);
            // Verify expected DWORD value (bit 6 set = 2^6 = 64 = 16#40)
            Assert.Equal(actual := result, expected := DWORD#16#0000_0040);

        END_METHOD

        {Test}
        METHOD PUBLIC TestOnlyUnholding
            VAR_TEMP
                result : DWORD;
            END_VAR

            ConfigureHoldCmdCfg(
                Starting := FALSE,
                Idle := FALSE,
                Suspended := FALSE,
                Execute := FALSE,
                Unholding := TRUE,
                Suspending := FALSE,
                Unsuspending := FALSE,
                Completing := FALSE,
                Completed := FALSE,
                holdCmdCfg => result);

            Assert.Equal(actual := result.%X12, expected := TRUE);
            Assert.Equal(actual := result.%X13, expected := FALSE);
            // Verify expected DWORD value (bit 12 set = 2^12 = 4096 = 16#1000)
            Assert.Equal(actual := result, expected := DWORD#16#0000_1000);

        END_METHOD

        {Test}
        METHOD PUBLIC TestOnlySuspending
            VAR_TEMP
                result : DWORD;
            END_VAR

            ConfigureHoldCmdCfg(
                Starting := FALSE,
                Idle := FALSE,
                Suspended := FALSE,
                Execute := FALSE,
                Unholding := FALSE,
                Suspending := TRUE,
                Unsuspending := FALSE,
                Completing := FALSE,
                Completed := FALSE,
                holdCmdCfg => result);

            Assert.Equal(actual := result.%X13, expected := TRUE);
            Assert.Equal(actual := result.%X12, expected := FALSE);
            Assert.Equal(actual := result.%X14, expected := FALSE);
            // Verify expected DWORD value (bit 13 set = 2^13 = 8192 = 16#2000)
            Assert.Equal(actual := result, expected := DWORD#16#0000_2000);

        END_METHOD

        {Test}
        METHOD PUBLIC TestOnlyUnsuspending
            VAR_TEMP
                result : DWORD;
            END_VAR

            ConfigureHoldCmdCfg(
                Starting := FALSE,
                Idle := FALSE,
                Suspended := FALSE,
                Execute := FALSE,
                Unholding := FALSE,
                Suspending := FALSE,
                Unsuspending := TRUE,
                Completing := FALSE,
                Completed := FALSE,
                holdCmdCfg => result);

            Assert.Equal(actual := result.%X14, expected := TRUE);
            Assert.Equal(actual := result.%X13, expected := FALSE);
            // Verify expected DWORD value (bit 14 set = 2^14 = 16384 = 16#4000)
            Assert.Equal(actual := result, expected := DWORD#16#0000_4000);

        END_METHOD

        {Test}
        METHOD PUBLIC TestOnlyCompleting
            VAR_TEMP
                result : DWORD;
            END_VAR

            ConfigureHoldCmdCfg(
                Starting := FALSE,
                Idle := FALSE,
                Suspended := FALSE,
                Execute := FALSE,
                Unholding := FALSE,
                Suspending := FALSE,
                Unsuspending := FALSE,
                Completing := TRUE,
                Completed := FALSE,
                holdCmdCfg => result);

            Assert.Equal(actual := result.%X16, expected := TRUE);
            Assert.Equal(actual := result.%X17, expected := FALSE);
            // Verify expected DWORD value (bit 16 set = 2^16 = 65536 = 16#10000)
            Assert.Equal(actual := result, expected := DWORD#16#0001_0000);

        END_METHOD

        {Test}
        METHOD PUBLIC TestOnlyCompleted
            VAR_TEMP
                result : DWORD;
            END_VAR

            ConfigureHoldCmdCfg(
                Starting := FALSE,
                Idle := FALSE,
                Suspended := FALSE,
                Execute := FALSE,
                Unholding := FALSE,
                Suspending := FALSE,
                Unsuspending := FALSE,
                Completing := FALSE,
                Completed := TRUE,
                holdCmdCfg => result);

            Assert.Equal(actual := result.%X17, expected := TRUE);
            Assert.Equal(actual := result.%X16, expected := FALSE);
            // Verify expected DWORD value (bit 17 set = 2^17 = 131072 = 16#20000)
            Assert.Equal(actual := result, expected := DWORD#16#0002_0000);

        END_METHOD

        {Test}
        METHOD PUBLIC TestANSICompliance_SuspendedAndExecute
            VAR_TEMP
                result : DWORD;
            END_VAR

            // Test the ANSI/ISA-TR88.00.02-2022 compliant configuration
            // Note: Only 'Suspended' and 'Execute' must be set for compliance
            ConfigureHoldCmdCfg(
                Starting := FALSE,
                Idle := FALSE,
                Suspended := TRUE,
                Execute := TRUE,
                Unholding := FALSE,
                Suspending := FALSE,
                Unsuspending := FALSE,
                Completing := FALSE,
                Completed := FALSE,
                holdCmdCfg => result);

            Assert.Equal(actual := result.%X5, expected := TRUE);   // Suspended
            Assert.Equal(actual := result.%X6, expected := TRUE);   // Execute
            Assert.Equal(actual := result.%X3, expected := FALSE);  // Starting
            Assert.Equal(actual := result.%X4, expected := FALSE);  // Idle

            // Verify expected DWORD value (bits 5+6 set = 32+64 = 96 = 16#60)
            Assert.Equal(actual := result, expected := DWORD#16#0000_0060);

        END_METHOD

        {Test}
        METHOD PUBLIC TestCombinationStartingAndIdle
            VAR_TEMP
                result : DWORD;
            END_VAR

            ConfigureHoldCmdCfg(
                Starting := TRUE,
                Idle := TRUE,
                Suspended := FALSE,
                Execute := FALSE,
                Unholding := FALSE,
                Suspending := FALSE,
                Unsuspending := FALSE,
                Completing := FALSE,
                Completed := FALSE,
                holdCmdCfg => result);

            Assert.Equal(actual := result.%X3, expected := TRUE);   // Starting
            Assert.Equal(actual := result.%X4, expected := TRUE);   // Idle
            Assert.Equal(actual := result.%X5, expected := FALSE);  // Suspended

            // Verify expected DWORD value (bits 3+4 set = 8+16 = 24 = 16#18)
            Assert.Equal(actual := result, expected := DWORD#16#0000_0018);

        END_METHOD

        {Test}
        METHOD PUBLIC TestCombinationHoldingStates
            VAR_TEMP
                result : DWORD;
            END_VAR

            // Test combination of holding-related states
            ConfigureHoldCmdCfg(
                Starting := FALSE,
                Idle := FALSE,
                Suspended := FALSE,
                Execute := FALSE,
                Unholding := TRUE,
                Suspending := TRUE,
                Unsuspending := TRUE,
                Completing := FALSE,
                Completed := FALSE,
                holdCmdCfg => result);

            Assert.Equal(actual := result.%X12, expected := TRUE);  // Unholding
            Assert.Equal(actual := result.%X13, expected := TRUE);  // Suspending
            Assert.Equal(actual := result.%X14, expected := TRUE);  // Unsuspending

            // Verify expected DWORD value (bits 12+13+14 set = 4096+8192+16384 = 28672 = 16#7000)
            Assert.Equal(actual := result, expected := DWORD#16#0000_7000);

        END_METHOD

        {Test}
        METHOD PUBLIC TestCombinationCompletingStates
            VAR_TEMP
                result : DWORD;
            END_VAR

            // Test combination of completing states
            ConfigureHoldCmdCfg(
                Starting := FALSE,
                Idle := FALSE,
                Suspended := FALSE,
                Execute := FALSE,
                Unholding := FALSE,
                Suspending := FALSE,
                Unsuspending := FALSE,
                Completing := TRUE,
                Completed := TRUE,
                holdCmdCfg => result);

            Assert.Equal(actual := result.%X16, expected := TRUE);  // Completing
            Assert.Equal(actual := result.%X17, expected := TRUE);  // Completed

            // Verify expected DWORD value (bits 16+17 set = 65536+131072 = 196608 = 16#30000)
            Assert.Equal(actual := result, expected := DWORD#16#0003_0000);

        END_METHOD

        {Test}
        METHOD PUBLIC TestAllStatesEnabled
            VAR_TEMP
                result : DWORD;
            END_VAR

            ConfigureHoldCmdCfg(
                Starting := TRUE,
                Idle := TRUE,
                Suspended := TRUE,
                Execute := TRUE,
                Unholding := TRUE,
                Suspending := TRUE,
                Unsuspending := TRUE,
                Completing := TRUE,
                Completed := TRUE,
                holdCmdCfg => result);

            // Verify all configured bits are set
            Assert.Equal(actual := result.%X3, expected := TRUE);   // Starting
            Assert.Equal(actual := result.%X4, expected := TRUE);   // Idle
            Assert.Equal(actual := result.%X5, expected := TRUE);   // Suspended
            Assert.Equal(actual := result.%X6, expected := TRUE);   // Execute
            Assert.Equal(actual := result.%X12, expected := TRUE);  // Unholding
            Assert.Equal(actual := result.%X13, expected := TRUE);  // Suspending
            Assert.Equal(actual := result.%X14, expected := TRUE);  // Unsuspending
            Assert.Equal(actual := result.%X16, expected := TRUE);  // Completing
            Assert.Equal(actual := result.%X17, expected := TRUE);  // Completed

            // Verify expected DWORD value (all configured bits set)
            // bits 3,4,5,6,12,13,14,16,17 = 8+16+32+64+4096+8192+16384+65536+131072 = 225400 = 16#37078
            Assert.Equal(actual := result, expected := DWORD#16#0003_7078);

        END_METHOD

        {Test}
        METHOD PUBLIC TestAllStatesDisabled
            VAR_TEMP
                result : DWORD;
            END_VAR

            ConfigureHoldCmdCfg(
                Starting := FALSE,
                Idle := FALSE,
                Suspended := FALSE,
                Execute := FALSE,
                Unholding := FALSE,
                Suspending := FALSE,
                Unsuspending := FALSE,
                Completing := FALSE,
                Completed := FALSE,
                holdCmdCfg => result);

            // Verify all configured bits are FALSE
            Assert.Equal(actual := result.%X3, expected := FALSE);
            Assert.Equal(actual := result.%X4, expected := FALSE);
            Assert.Equal(actual := result.%X5, expected := FALSE);
            Assert.Equal(actual := result.%X6, expected := FALSE);
            Assert.Equal(actual := result.%X12, expected := FALSE);
            Assert.Equal(actual := result.%X13, expected := FALSE);
            Assert.Equal(actual := result.%X14, expected := FALSE);
            Assert.Equal(actual := result.%X16, expected := FALSE);
            Assert.Equal(actual := result.%X17, expected := FALSE);

            // Verify expected DWORD value (no bits set = 0)
            Assert.Equal(actual := result, expected := DWORD#16#0000_0000);

        END_METHOD

        {Test}
        METHOD PUBLIC TestUnusedBitsRemainZero
            VAR_TEMP
                result : DWORD;
            END_VAR

            // Test with all configurable states enabled
            ConfigureHoldCmdCfg(
                Starting := TRUE,
                Idle := TRUE,
                Suspended := TRUE,
                Execute := TRUE,
                Unholding := TRUE,
                Suspending := TRUE,
                Unsuspending := TRUE,
                Completing := TRUE,
                Completed := TRUE,
                holdCmdCfg => result);

            // Test that unused bits remain 0
            Assert.Equal(actual := result.%X0, expected := FALSE);   // Unused
            Assert.Equal(actual := result.%X1, expected := FALSE);   // Unused
            Assert.Equal(actual := result.%X2, expected := FALSE);   // Unused
            Assert.Equal(actual := result.%X7, expected := FALSE);   // Unused
            Assert.Equal(actual := result.%X8, expected := FALSE);   // Unused
            Assert.Equal(actual := result.%X9, expected := FALSE);   // Unused
            Assert.Equal(actual := result.%X10, expected := FALSE);  // Unused
            Assert.Equal(actual := result.%X11, expected := FALSE);  // Unused
            Assert.Equal(actual := result.%X15, expected := FALSE);  // Unused
            Assert.Equal(actual := result.%X18, expected := FALSE);  // Unused
            Assert.Equal(actual := result.%X31, expected := FALSE);  // Unused (MSB)

        END_METHOD

        {Test}
        METHOD PUBLIC TestBitMappingVerification
            VAR_TEMP
                result : DWORD;
            END_VAR

            // Test specific bit mappings one by one

            // Test Starting -> bit 3
            ConfigureHoldCmdCfg(
                Starting := TRUE,
                Idle := FALSE, Suspended := FALSE, Execute := FALSE,
                Unholding := FALSE, Suspending := FALSE, Unsuspending := FALSE,
                Completing := FALSE, Completed := FALSE,
                holdCmdCfg => result);
            Assert.Equal(actual := result.%X3, expected := TRUE);
            Assert.Equal(actual := result, expected := DWORD#16#0000_0008);

            // Test Idle -> bit 4
            ConfigureHoldCmdCfg(
                Starting := FALSE,
                Idle := TRUE, Suspended := FALSE, Execute := FALSE,
                Unholding := FALSE, Suspending := FALSE, Unsuspending := FALSE,
                Completing := FALSE, Completed := FALSE,
                holdCmdCfg => result);
            Assert.Equal(actual := result.%X4, expected := TRUE);
            Assert.Equal(actual := result, expected := DWORD#16#0000_0010);

            // Test Unholding -> bit 12
            ConfigureHoldCmdCfg(
                Starting := FALSE, Idle := FALSE, Suspended := FALSE, Execute := FALSE,
                Unholding := TRUE,
                Suspending := FALSE, Unsuspending := FALSE,
                Completing := FALSE, Completed := FALSE,
                holdCmdCfg => result);
            Assert.Equal(actual := result.%X12, expected := TRUE);
            Assert.Equal(actual := result, expected := DWORD#16#0000_1000);

        END_METHOD

        {Test}
        METHOD PUBLIC TestHighOrderBitMapping
            VAR_TEMP
                result : DWORD;
            END_VAR

            // Test high-order bit mappings (Completing and Completed)
            ConfigureHoldCmdCfg(
                Starting := FALSE, Idle := FALSE, Suspended := FALSE, Execute := FALSE,
                Unholding := FALSE, Suspending := FALSE, Unsuspending := FALSE,
                Completing := TRUE,
                Completed := FALSE,
                holdCmdCfg => result);

            Assert.Equal(actual := result.%X16, expected := TRUE);  // Completing -> bit 16
            Assert.Equal(actual := result.%X17, expected := FALSE); // Completed -> bit 17
            Assert.Equal(actual := result, expected := DWORD#16#0001_0000);

            // Test Completed -> bit 17
            ConfigureHoldCmdCfg(
                Starting := FALSE, Idle := FALSE, Suspended := FALSE, Execute := FALSE,
                Unholding := FALSE, Suspending := FALSE, Unsuspending := FALSE,
                Completing := FALSE,
                Completed := TRUE,
                holdCmdCfg => result);

            Assert.Equal(actual := result.%X16, expected := FALSE); // Completing -> bit 16
            Assert.Equal(actual := result.%X17, expected := TRUE);  // Completed -> bit 17
            Assert.Equal(actual := result, expected := DWORD#16#0002_0000);

        END_METHOD

        {Test}
        METHOD PUBLIC TestANSI_ExtendedCompliance
            VAR_TEMP
                result : DWORD;
            END_VAR

            // Test ANSI compliance with additional commonly used states
            ConfigureHoldCmdCfg(
                Starting := TRUE,
                Idle := TRUE,
                Suspended := TRUE,  // Required for ANSI compliance
                Execute := TRUE,    // Required for ANSI compliance
                Unholding := FALSE,
                Suspending := FALSE,
                Unsuspending := FALSE,
                Completing := FALSE,
                Completed := FALSE,
                holdCmdCfg => result);

            // Verify ANSI required states
            Assert.Equal(actual := result.%X5, expected := TRUE);   // Suspended (ANSI required)
            Assert.Equal(actual := result.%X6, expected := TRUE);   // Execute (ANSI required)

            // Verify additional states
            Assert.Equal(actual := result.%X3, expected := TRUE);   // Starting
            Assert.Equal(actual := result.%X4, expected := TRUE);   // Idle

            // Verify expected DWORD value (bits 3+4+5+6 set = 8+16+32+64 = 120 = 16#78)
            Assert.Equal(actual := result, expected := DWORD#16#0000_0078);

        END_METHOD

    END_CLASS

END_NAMESPACE
